{attribute 'GeneratedUsingTerminal: EK1122-0000-0018'}
{attribute addProperty BoxType "EK1122-0000-0018"}
{attribute addProperty Id "Beckhoff_ER3xxxsub_EK1100EK1100_AB5A94672A_0001_ER3174_0002_0016ER3174_0E4717A052A_0002_ER3174_0002_0022ER3174_0E4717A052A_0003_ER3174_0002_0023ER3174_0E4717A052A_0004_ER3184_0002_0019ER3184_0E4717A052A_0005_ER3184_0002_0020ER3184_0E4717A052A_0006_ER3184_0002_0021ER3184_0E4717A052A_0007_ER3184_1002_0020ER3184_0E4717A052A_0008_ER3184_1002_0021ER3184_0E4717A052A_0009_ER3204_0002_0016ER3204_7A00DD1E52A_0010_ER3204_0002_0020ER3204_7A00DD1E52A_0011_ER3204_0002_0021ER3204_BF0B7ECE48A_0012_ER3314_0002_0021ER3314_6BF23D5548"}
{attribute addProperty CRC "1219793750"}
{attribute addProperty Size "618"}
TYPE Beckhoff_ER3xxxEK1122_48B49356 EXTENDS EK1122_AB5A9467 :
STRUCT
	{attribute addProperty Name "Beckhoff_ER3xxxsub_EK1100"}
	Beckhoff_ER3xxxsub_EK1100 : EK1100_AB5A9467;
	{attribute addProperty Name "A_0001_ER3174_0002_0016"}
	A_0001_ER3174_0002_0016 : ER3174_0E4717A0;
	{attribute addProperty Name "A_0002_ER3174_0002_0022"}
	A_0002_ER3174_0002_0022 : ER3174_0E4717A0;
	{attribute addProperty Name "A_0003_ER3174_0002_0023"}
	A_0003_ER3174_0002_0023 : ER3174_0E4717A0;
	{attribute addProperty Name "A_0004_ER3184_0002_0019"}
	A_0004_ER3184_0002_0019 : ER3184_0E4717A0;
	{attribute addProperty Name "A_0005_ER3184_0002_0020"}
	A_0005_ER3184_0002_0020 : ER3184_0E4717A0;
	{attribute addProperty Name "A_0006_ER3184_0002_0021"}
	A_0006_ER3184_0002_0021 : ER3184_0E4717A0;
	{attribute addProperty Name "A_0007_ER3184_1002_0020"}
	A_0007_ER3184_1002_0020 : ER3184_0E4717A0;
	{attribute addProperty Name "A_0008_ER3184_1002_0021"}
	A_0008_ER3184_1002_0021 : ER3184_0E4717A0;
	{attribute addProperty Name "A_0009_ER3204_0002_0016"}
	A_0009_ER3204_0002_0016 : ER3204_7A00DD1E;
	{attribute addProperty Name "A_0010_ER3204_0002_0020"}
	A_0010_ER3204_0002_0020 : ER3204_7A00DD1E;
	{attribute addProperty Name "A_0011_ER3204_0002_0021"}
	A_0011_ER3204_0002_0021 : ER3204_BF0B7ECE;
	{attribute addProperty Name "A_0012_ER3314_0002_0021"}
	A_0012_ER3314_0002_0021 : ER3314_6BF23D55;
END_STRUCT
END_TYPE

(* stored: Version 1.2.0.0, ProductVersion 3.1.4024.9
   DUT Beckhoff_ER3xxxEK1122_48B49356: Id {31715521-8128-47d8-8b70-3a9a7739cb1f} *)
